// TIA Portal V16 export
// export: Created 2021-07-12T14:47:19.7297692Z, ExportSetting WithDefaults, DisplayName Totally Integrated Automation Portal, DisplayVersion V16, DisplayName TIA Portal Version Control Interface, DisplayVersion V16, DisplayName TIA Portal Openness, DisplayVersion V16, DisplayName STEP 7 Professional, DisplayVersion V16, DisplayName STEP 7 Safety, DisplayVersion V16, DisplayName WinCC Professional, DisplayVersion V16
TYPE "LSimaHydTO_typeDynamicAxisModel"
TITLE = LSimaHydTO_typeDynamicAxisModel
// Settings of the balancing filter
// stored: IsFailsafeCompliant false
   STRUCT
      VelocityTimeConstant { S7_SetPoint := 'True'} : LReal;   // Speed control loop substitute time [s]
      ForceTimeConstant { S7_SetPoint := 'True'} : LReal;   // Force control loop substitute time [s]
   END_STRUCT;
END_TYPE
